{attribute addProperty BoxType "EL3001-0000-0017"}
{attribute addProperty Id "StatusAT %I*Status_C6F82E6F658.1251ValueAT %I*INT16217"}
{attribute addProperty CRC "3038476796"}
{attribute addProperty SizeInBites "81"}
{attribute addProperty SizeInBytes "10.125"}
TYPE AI_Standard_B51B79FC :
STRUCT
	{attribute addProperty Name "Status"}
	Status AT %I* : Status_C6F82E6F;
	{attribute addProperty Name "Value"}
	Value AT %I* : INT;
END_STRUCT
END_TYPE

(* stored: Version 1.2.0.0, ProductVersion 3.1.4024.9
   DUT AI_Standard_B51B79FC: Id {56a2d871-9b96-4110-9720-86532b73f7bc} *)
